// Mitsubishi GX Works2 project: 14-06-2020 LAB 2_Sequence_STL   PLC: FX3G

PROGRAM MAIN
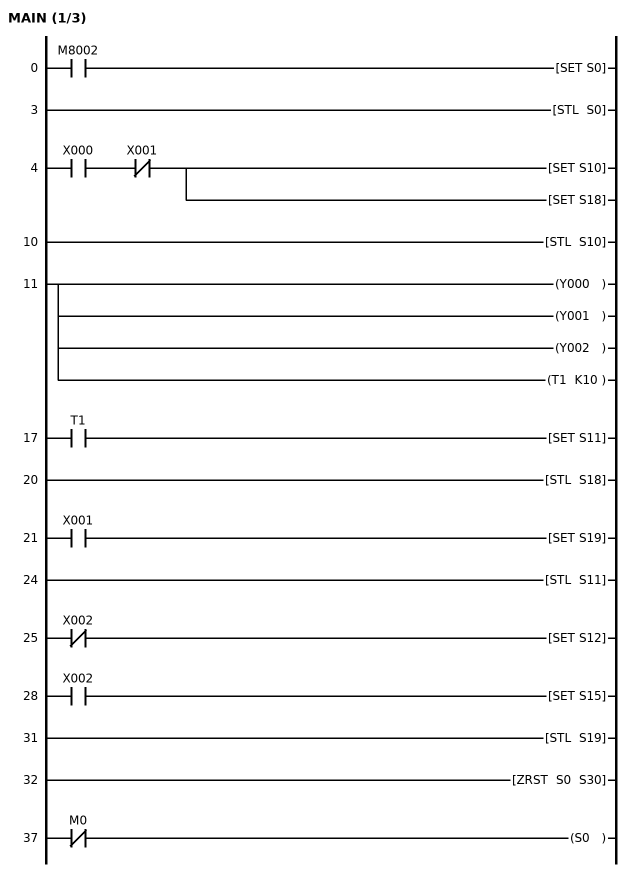
0     LD      M8002
      SET     S0
3     STL     S0
4     LD      X000
      ANI     X001
      SET     S10
      SET     S18
10    STL     S10
11    OUT     Y000
      OUT     Y001
      OUT     Y002
      OUT     T1 K10
17    LD      T1
      SET     S11
20    STL     S18
21    LD      X001
      SET     S19
24    STL     S11
25    LDI     X002
      SET     S12
28    LD      X002
      SET     S15
31    STL     S19
32    ZRST    S0 S30
37    LDI     M0
      OUT     S0
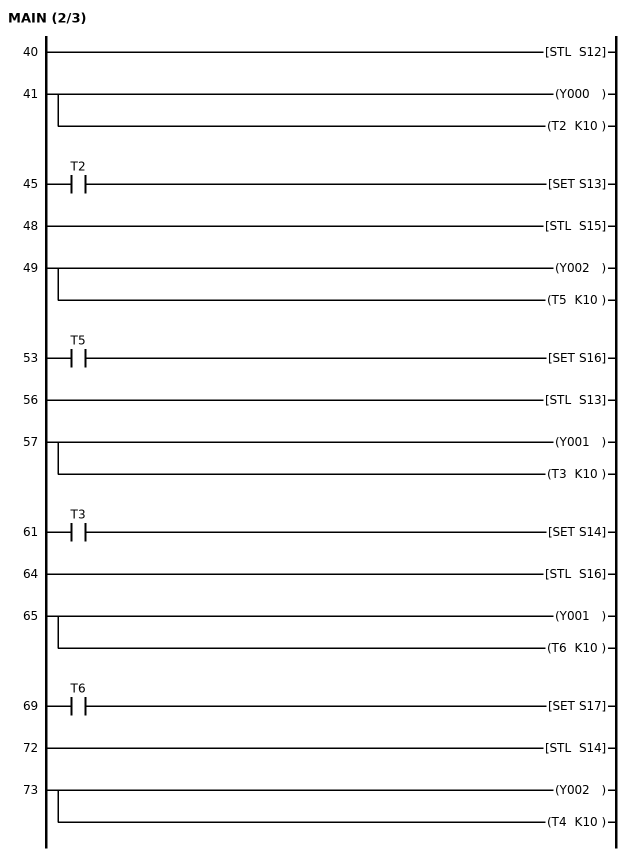
40    STL     S12
41    OUT     Y000
      OUT     T2 K10
45    LD      T2
      SET     S13
48    STL     S15
49    OUT     Y002
      OUT     T5 K10
53    LD      T5
      SET     S16
56    STL     S13
57    OUT     Y001
      OUT     T3 K10
61    LD      T3
      SET     S14
64    STL     S16
65    OUT     Y001
      OUT     T6 K10
69    LD      T6
      SET     S17
72    STL     S14
73    OUT     Y002
      OUT     T4 K10
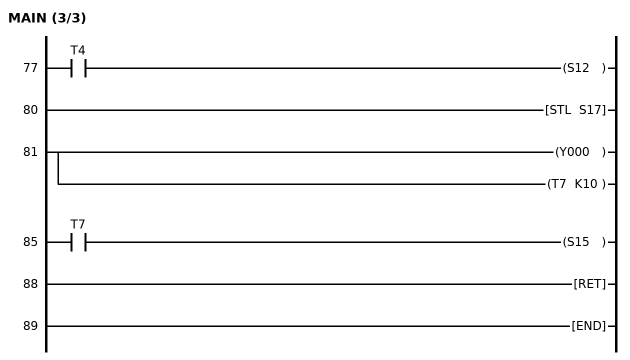
77    LD      T4
      OUT     S12
80    STL     S17
81    OUT     Y000
      OUT     T7 K10
85    LD      T7
      OUT     S15
88    RET
89    END
END_PROGRAM
